TYPE Parameters_Typ :
STRUCT
	//TimerPressDown1:DINT;//[MS]
	
	Continues:BOOL;
	NumberOfCycles:UDINT;
	WebLinarSpeed:LREAL;//[mm]
	WebLinarSpeedSlow:LREAL;//[mm]
	
	DancerFillSpeed :LREAL;//[Degrees per seconds]
	
	
	
	MotorVelocity :INT;
	DistanceToMove:UINT;
	
	
	OutGripperEndPosition:LREAL;
	OutGripperHomeVelocity:LREAL;
	OutGripperProcessVelocity:LREAL;
	
	
	UW_1_Param	: UnwinderParameters_Typ;
	UW_2_Param	: UnwinderParameters_Typ;
	
END_STRUCT
END_TYPE

(* stored: Version 1.1.0.1, ProductVersion 3.1.4024.3
   DUT Parameters_Typ: Id {fefcba5b-ea80-4050-ab7b-7404de5956b7} *)
